FUNCTION_BLOCK FB_Machine_Run EXTENDS CycleHandleFB
VAR_INPUT
	Ctrl_ref:					REFERENCE TO Ctrl_Typ;
	 FB_RW_Ctrl_ref:			REFERENCE TO FB_RW_Ctrl;
END_VAR
VAR_OUTPUT
END_VAR
VAR
	MethInitDone:		BOOL;
	FB_HeaterProtection:FB_HeaterProtection;
END_VAR
VAR CONSTANT

// States are global
(*		
	MACHINE_RUN_INIT:						INT:=0;
	MACHINE_COLD_CUT_VALVE_OPEN:			INT:=10;
	MACHINE_WELD_VALVE_OPEN:				INT:=20;	
	MACHINE_HEATER_ON:						INT:=30;	
	MACHINE_HEATER_OFF:						INT:=40;
	MACHINE_VALVE_CLOSE:					INT:=50;	
	MACHINE_DONE:							INT:=100;	

*)

END_VAR

	IF NOT MethInitDone THEN
		MethInitDone	:= Meth_Init();
	END_IF
	
	
	IF  THIS^.CMD.Pause = FALSE THEN
		
		//-----------------------------
		//State Machine
		//-----------------------------
		CASE THIS^.StepNo OF
			MACHINE_RUN_INIT:
				IF THIS^.StepOneShotTrig THEN
					THIS^.Monitoring.StepMessage	:= 'Init: Start.';
					THIS^.Delay(IN:=FALSE);
					Meth_Rest_IO();
				ELSIF Meth_Enable(TRUE) THEN
					THIS^.StepNo	:= 	MACHINE_WAIT_DANCER_FULL;
				//	THIS^.StepNo	:= 	MACHINE_GRIPPER_END_POSITION;
				END_IF								
			
				
			MACHINE_WAIT_DANCER_FULL:
				IF THIS^.StepOneShotTrig THEN
					THIS^.Monitoring.StepMessage	:= 'Wait Dancer full';
					THIS^.Delay(IN:=FALSE);
				ELSIF Meth_WaitDancerFull(TRUE) THEN
					THIS^.StepNo	:= 	MACHINE_GRIPPER_RETRACT;
				END_IF					
								
	
			MACHINE_GRIPPER_RETRACT:
				IF THIS^.StepOneShotTrig THEN
					THIS^.Monitoring.StepMessage	:= 'Gripper retract';
					THIS^.Delay(IN:=FALSE);
					
				ELSIF Meth_gripperRetract(TRUE) THEN
					THIS^.StepNo	:= 	MACHINE_GRIPPER_END_POSITION;
				END_IF	

									
			MACHINE_GRIPPER_END_POSITION:
				IF THIS^.StepOneShotTrig THEN
					THIS^.Monitoring.StepMessage	:= 'Machine WAIT position';
					THIS^.Delay(IN:=FALSE);
				ELSIF Meth_gripperEndPosition(TRUE) THEN
					THIS^.StepNo	:= 	MACHINE_OUT_GRIPPER_START_POSITION;
				END_IF					
			
			MACHINE_OUT_GRIPPER_START_POSITION:
				IF THIS^.StepOneShotTrig THEN
					THIS^.Monitoring.StepMessage	:= 'Output Grippers to start position';
					Meth_OutGripperStartPos(FALSE) ;
				ELSIF Meth_OutGripperStartPos(TRUE) THEN
					THIS^.StepNo	:= 	MACHINE_OUT_GRIPPER_CLAMP;
				END_IF				
							
				
			MACHINE_OUT_GRIPPER_CLAMP:
				IF THIS^.StepOneShotTrig THEN
					THIS^.Monitoring.StepMessage	:= 'Machine grippers clamp';
					THIS^.Delay(IN:=FALSE);
				ELSIF Meth_OutGripperClamp(TRUE) THEN
					THIS^.StepNo	:= 	MACHINE_GRIPPER_OPEN;
				END_IF	
			

			MACHINE_GRIPPER_OPEN:
				IF THIS^.StepOneShotTrig THEN
					THIS^.Monitoring.StepMessage	:= 'Gripper Open';
					THIS^.Delay(IN:=FALSE);
				ELSIF Meth_gripperOpen(TRUE) THEN
					THIS^.StepNo	:= 	MACHINE_GRIPPER_START_POSITION;
				END_IF					
						
				
			MACHINE_GRIPPER_START_POSITION:
				IF THIS^.StepOneShotTrig THEN
					THIS^.Monitoring.StepMessage	:= 'Machine start position';
					THIS^.Delay(IN:=FALSE);
					
				ELSIF Meth_gripperStartPosition(TRUE) THEN
					THIS^.StepNo	:= 	MACHINE_GRIPPER_EXCTRACT;
				END_IF	
	
			
			MACHINE_GRIPPER_EXCTRACT:
			IF THIS^.StepOneShotTrig THEN
				THIS^.Monitoring.StepMessage	:= 'Gripper Extract';
				THIS^.Delay(IN:=FALSE);
			ELSIF Meth_gripperExtract(TRUE) THEN
				THIS^.StepNo	:= 	MACHINE_GRIPPER_CLOSE;
			END_IF				
				
			MACHINE_GRIPPER_CLOSE:
				IF THIS^.StepOneShotTrig THEN
					THIS^.Monitoring.StepMessage	:= 'Gripper Close';
					THIS^.Delay(IN:=FALSE);
				ELSIF Meth_gripperClose(TRUE) THEN
					THIS^.StepNo	:= 	MACHINE_COLD_CUT_VALVE_OPEN;
				END_IF	
	
			MACHINE_COLD_CUT_VALVE_OPEN:
				IF THIS^.StepOneShotTrig THEN
					THIS^.Monitoring.StepMessage	:= 'Cold cut valve open';
					THIS^.Delay(IN:=FALSE);
				ELSIF Meth_ColdCutValveOpen(TRUE) THEN
					THIS^.StepNo	:= 	MACHINE_WELD_VALVE_OPEN;
				END_IF	

			MACHINE_WELD_VALVE_OPEN://and gripper open
				IF THIS^.StepOneShotTrig THEN
					THIS^.Monitoring.StepMessage	:= 'Hot weld valve open press Down';
					THIS^.Delay(IN:=FALSE);
				ELSIF Meth_HotWeldValveOpen(TRUE) THEN
					THIS^.StepNo	:= 	MACHINE_HEATER_ON;
				END_IF					
				
			MACHINE_HEATER_ON://
				IF THIS^.StepOneShotTrig THEN
					THIS^.Monitoring.StepMessage	:= 'Heater ON';
					THIS^.Delay(IN:=FALSE);
				ELSIF Meth_HeaterON(TRUE) THEN
					THIS^.StepNo	:= 	MACHINE_HEATER_OFF;
				END_IF								
				
			MACHINE_HEATER_OFF://gripper retract
				IF THIS^.StepOneShotTrig THEN
					THIS^.Monitoring.StepMessage	:= 'Heater Off';
					THIS^.Delay(IN:=FALSE);
				ELSIF Meth_HeaterOff(TRUE) THEN
					THIS^.StepNo	:= 	MACHINE_CUT_WEB;
				END_IF					
						
			MACHINE_CUT_WEB:
				IF THIS^.StepOneShotTrig THEN
					THIS^.Monitoring.StepMessage	:= 'Close valves';
					THIS^.Delay(IN:=FALSE);
					gMachineCtrl.IO.Out.KniveCut:=NOT(gMachineCtrl.IO.Out.KniveCut);
				ELSIF Meth_CutWeb(TRUE) THEN
					THIS^.StepNo	:= 	MACHINE_VALVE_CLOSE;
				END_IF		
				
			MACHINE_VALVE_CLOSE:
				IF THIS^.StepOneShotTrig THEN
					THIS^.Monitoring.StepMessage	:= 'Close valves';
					THIS^.Delay(IN:=FALSE);
				ELSIF Meth_HeaterValvesClose(TRUE) THEN
					THIS^.StepNo	:= 	MACHINE_OUT_GRIPPER_END_POSITION;
				END_IF					
				
			MACHINE_OUT_GRIPPER_END_POSITION:
				IF THIS^.StepOneShotTrig THEN
					THIS^.Monitoring.StepMessage	:= 'Output Grippers to start position';
					Meth_OutGripperEndPos(FALSE) ;
				ELSIF Meth_OutGripperEndPos(TRUE) THEN
					THIS^.StepNo	:= 	MACHINE_DONE;
				END_IF								
				
			MACHINE_DONE:
				IF THIS^.StepOneShotTrig THEN
					THIS^.Monitoring.StepMessage	:= 'Machine cycle Done';
				ELSIF Meth_Done(TRUE) THEN
					THIS^.StepNo	:= 	MACHINE_RUN_INIT;
				END_IF			
			
				
			//UnUsed	
			
								
		END_CASE
	
	ELSE
		THIS^.Monitoring.StepMessage:= 'Pause';
		
		IF THIS^.Status.Fault = TRUE THEN
		//IF Meth_EmStop(TRUE) THEN
				THIS^.CMD.ResetCycle	:= TRUE;		// Reset the all state machine to start point
		//END_IF
			
		END_IF
		
	END_IF
	
	//============================================================================================
	// Reset Internal Function Blocks
	IF THIS^.CMD.ResetCycle = TRUE THEN
		IF FB_RW_Ctrl_ref.Running OR FB_RW_Ctrl_ref.Pause OR FB_RW_Ctrl_ref.Fault THEN
			FB_RW_Ctrl_ref.ResetCycle	:= TRUE;
		END_IF
	END_IF	
	
	THIS^.FB_HeaterProtection();
	THIS^.Delay();
	THIS^.CH_Logic();
	
	// Reset Meth_EmStop when at Init State
	IF THIS^.Pause = FALSE THEN
		//Meth_EmStop(FALSE);
	END_IF

METHOD PRIVATE Meth_ColdCutValveOpen : BOOL
VAR_INPUT
	Execute: 	BOOL;
END_VAR


	THIS^.Monitoring.StepMessage			:= 'Cold Cut Valve Open';
	THIS^.Monitoring.Error_Text				:= ' Fail';
	//THIS^.CMD.Deacivate_Sequence_Time_Out	:= TRUE;	// Disable time out to the all sequence
	THIS^.CMD.DeactivateStepTimeOut			:= TRUE;	// Disable time out to the actual step
	THIS^.Parameter.TimeOut					:= T#5S;


	
	gMachineCtrl.IO.Out.Buzzer	:=TRUE;
										
	THIS^.Delay.IN:=TRUE;
	THIS^.Delay.PT :=DINT_TO_TIME( Persist.PersistentStruct.TimeColdCutPressDown);// Ctrl_ref.Parameters.TimerPressDown1);
	IF THIS^.Delay.Q THEN
		Meth_ColdCutValveOpen	:= TRUE;
		gMachineCtrl.IO.Out.GripperOpen:=TRUE;
	END_IF
END_METHOD

METHOD Meth_CutWeb : BOOL
VAR_INPUT
	Execute: 	BOOL;
END_VAR
	THIS^.Monitoring.StepMessage			:= 'Cut Web';
	THIS^.Monitoring.Error_Text				:= ' Fail';
	//THIS^.CMD.Deacivate_Sequence_Time_Out	:= TRUE;	// Disable time out to the all sequence
	THIS^.CMD.DeactivateStepTimeOut			:= TRUE;	// Disable time out to the actual step
	THIS^.Parameter.TimeOut					:= T#5S;

	
											
	THIS^.Delay.IN:=TRUE;
	THIS^.Delay.PT :=DINT_TO_TIME( Persist.PersistentStruct.TimeKniveVut);// Ctrl_ref.Parameters.TimerPressDown1);
	IF THIS^.Delay.Q THEN
		Meth_CutWeb	:= TRUE;
		
		//gMachineCtrl.Parameters.UW_1_Param.EnableTension:=TRUE;
		//gMachineCtrl.Parameters.UW_2_Param.EnableTension:=TRUE;
		
	END_IF
END_METHOD

METHOD PRIVATE Meth_Done : BOOL
VAR_INPUT
	Execute: 	BOOL;
END_VAR


	//THIS^.Monitoring.StepMessage			:= 'Press 1 engage';
	//THIS^.Monitoring.Error_Text				:= 'Press 1 engage Fail';
	//THIS^.CMD.Deacivate_Sequence_Time_Out	:= TRUE;	// Disable time out to the all sequence
	//THIS^.CMD.DeactivateStepTimeOut			:= TRUE;	// Disable time out to the actual step
	//THIS^.Parameter.TimeOut					:= T#5S;

	//gMachineCtrl.Parameters.UW_1_Param.EnableDancer :=FALSE;
	//gMachineCtrl.Parameters.UW_2_Param.EnableDancer:=FALSE;	
	
	THIS^.Status.Done		:= TRUE;
	THIS^.Status.Running	:= FALSE;									
	Meth_Done	:= TRUE;
END_METHOD

METHOD PRIVATE Meth_Enable : BOOL
VAR_INPUT
	Execute: 	BOOL;
END_VAR


IF THIS^.CMD.Start THEN
	
	THIS^.Monitoring.StepMessage			:= 'Start';
	THIS^.Monitoring.Error_Text				:= 'Start Fail';
	THIS^.CMD.Deacivate_Sequence_Time_Out	:= TRUE;	// Disable time out to the all sequence
	THIS^.CMD.DeactivateStepTimeOut			:= TRUE;	// Disable time out to the actual step
	THIS^.Parameter.TimeOut					:= T#0.5S;

	THIS^.CMD.Start			:= FALSE;
	THIS^.Status.Done		:= FALSE;
	THIS^.Status.Running	:= TRUE;
	
	// Reset Commands and Statuses												
	
	Meth_Enable	:= TRUE;
END_IF
END_METHOD

METHOD PRIVATE Meth_gripperClose : BOOL
VAR_INPUT
	Execute: 	BOOL;
END_VAR


	THIS^.Monitoring.StepMessage			:= 'Gripper Close';
	THIS^.Monitoring.Error_Text				:= ' Fail';
	//THIS^.CMD.Deacivate_Sequence_Time_Out	:= TRUE;	// Disable time out to the all sequence
	THIS^.CMD.DeactivateStepTimeOut			:= TRUE;	// Disable time out to the actual step
	THIS^.Parameter.TimeOut					:= T#5S;

	gMachineCtrl.IO.Out.GripperOpen:=TRUE;
											
	THIS^.Delay.IN:=TRUE;
	THIS^.Delay.PT :=DINT_TO_TIME( Persist.PersistentStruct.TimeGripperOpen);// Ctrl_ref.Parameters.TimerPressDown1);
	IF THIS^.Delay.Q THEN
		Meth_gripperClose	:= TRUE;
		
		//gMachineCtrl.Parameters.UW_1_Param.EnableTension:=TRUE;
		//gMachineCtrl.Parameters.UW_2_Param.EnableTension:=TRUE;
		
	END_IF
END_METHOD

METHOD PRIVATE Meth_gripperEndPosition : BOOL
VAR_INPUT
	Execute: 	BOOL;
END_VAR


	//THIS^.Monitoring.StepMessage			:= 'GripperStartPosition';
	THIS^.Monitoring.Error_Text				:= ' Fail';
	//THIS^.CMD.Deacivate_Sequence_Time_Out	:= TRUE;	// Disable time out to the all sequence
	THIS^.CMD.DeactivateStepTimeOut			:= TRUE;	// Disable time out to the actual step
	THIS^.Parameter.TimeOut					:= T#5S;

	gMachineCtrl.IO.Out.GripperPistonPosition:=TRUE;
	
	gMachineCtrl.IO.Out.ExternalNipMotor:=TRUE;
		
	//gMachineCtrl.Parameters.UW_1_Param.kp := gMachineCtrl.Parameters.UW_1_Param.kpMove;
	////gMachineCtrl.Parameters.UW_1_Param.TN := gMachineCtrl.Parameters.UW_1_Param.TNMove;
	//.Parameters.UW_2_Param.kp := gMachineCtrl.Parameters.UW_2_Param.kpMove;
	//gMachineCtrl.Parameters.UW_2_Param.TN := gMachineCtrl.Parameters.UW_2_Param.TNMove;



							
	THIS^.Delay.IN:=TRUE;
	THIS^.Delay.PT :=DINT_TO_TIME( Persist.PersistentStruct.TimeGripperStartPosition);// Ctrl_ref.Parameters.TimerPressDown1);
	IF THIS^.Delay.Q THEN
		Meth_gripperEndPosition	:= TRUE;
		
	//.Parameters.UW_1_Param.kp := 0.1;
	//gMachineCtrl.Parameters.UW_1_Param.TN := T#0MS;
	//gMachineCtrl.Parameters.UW_2_Param.kp := 0.1;
	//gMachineCtrl.Parameters.UW_2_Param.TN := T#0MS;			
	
	gMachineCtrl.IO.Out.ExternalNipMotor:=FALSE;
		
	END_IF
END_METHOD

METHOD PRIVATE Meth_gripperExtract : BOOL
VAR_INPUT
	Execute: 	BOOL;
END_VAR


	//THIS^.Monitoring.StepMessage			:= 'Gripper Retract';
	THIS^.Monitoring.Error_Text				:= ' Fail';
	//THIS^.CMD.Deacivate_Sequence_Time_Out	:= TRUE;	// Disable time out to the all sequence
	THIS^.CMD.DeactivateStepTimeOut			:= TRUE;	// Disable time out to the actual step
	THIS^.Parameter.TimeOut					:= T#5S;

	gMachineCtrl.IO.Out.GripperRetract:=TRUE;
											
	THIS^.Delay.IN:=TRUE;
	THIS^.Delay.PT :=DINT_TO_TIME( Persist.PersistentStruct.TimeGripperRetract);// Ctrl_ref.Parameters.TimerPressDown1);
	IF THIS^.Delay.Q THEN
		Meth_gripperExtract	:= TRUE;
	END_IF
END_METHOD

METHOD PRIVATE Meth_gripperOpen : BOOL
VAR_INPUT
	Execute: 	BOOL;
END_VAR


	//THIS^.Monitoring.StepMessage			:= 'Gripper Open';
	THIS^.Monitoring.Error_Text				:= ' Fail';
	//THIS^.CMD.Deacivate_Sequence_Time_Out	:= TRUE;	// Disable time out to the all sequence
	THIS^.CMD.DeactivateStepTimeOut			:= TRUE;	// Disable time out to the actual step
	THIS^.Parameter.TimeOut					:= T#5S;

	gMachineCtrl.IO.Out.GripperOpen:=FALSE;
											
	THIS^.Delay.IN:=TRUE;
	THIS^.Delay.PT :=DINT_TO_TIME( Persist.PersistentStruct.TimeGripperOpen);// Ctrl_ref.Parameters.TimerPressDown1);
	IF THIS^.Delay.Q THEN
		Meth_gripperOpen	:= TRUE;
	END_IF
END_METHOD

METHOD PRIVATE Meth_gripperRetract : BOOL
VAR_INPUT
	Execute: 	BOOL;
END_VAR


	//THIS^.Monitoring.StepMessage			:= 'Gripper Retract';
	THIS^.Monitoring.Error_Text				:= ' Fail';
	//THIS^.CMD.Deacivate_Sequence_Time_Out	:= TRUE;	// Disable time out to the all sequence
	THIS^.CMD.DeactivateStepTimeOut			:= TRUE;	// Disable time out to the actual step
	THIS^.Parameter.TimeOut					:= T#5S;

	gMachineCtrl.IO.Out.GripperRetract:=FALSE;
											
	THIS^.Delay.IN:=TRUE;
	THIS^.Delay.PT :=DINT_TO_TIME( Persist.PersistentStruct.TimeGripperRetract);// Ctrl_ref.Parameters.TimerPressDown1);
	IF THIS^.Delay.Q THEN
		Meth_gripperRetract	:= TRUE;
	END_IF
END_METHOD

METHOD PRIVATE Meth_gripperStartPosition : BOOL
VAR_INPUT
	Execute: 	BOOL;
END_VAR


	//THIS^.Monitoring.StepMessage			:= 'GripperStartPosition';
	THIS^.Monitoring.Error_Text				:= ' Fail';
	//THIS^.CMD.Deacivate_Sequence_Time_Out	:= TRUE;	// Disable time out to the all sequence
	THIS^.CMD.DeactivateStepTimeOut			:= TRUE;	// Disable time out to the actual step
	THIS^.Parameter.TimeOut					:= T#5S;

	gMachineCtrl.IO.Out.GripperPistonPosition:=FALSE;
											
	THIS^.Delay.IN:=TRUE;
	THIS^.Delay.PT :=DINT_TO_TIME( Persist.PersistentStruct.TimeGripperHomePosition);// Ctrl_ref.Parameters.TimerPressDown1);
	IF THIS^.Delay.Q THEN
		Meth_gripperStartPosition	:= TRUE;
	END_IF
END_METHOD

METHOD PRIVATE Meth_HeaterOff : BOOL
VAR_INPUT
	Execute: 	BOOL;
END_VAR


	THIS^.Monitoring.StepMessage			:= 'Heater Off';
	THIS^.Monitoring.Error_Text				:= ' Heater Off Fail';
	//THIS^.CMD.Deacivate_Sequence_Time_Out	:= TRUE;	// Disable time out to the all sequence
	THIS^.CMD.DeactivateStepTimeOut			:= TRUE;	// Disable time out to the actual step
	THIS^.Parameter.TimeOut					:= T#5S;

	
											
	THIS^.Delay.IN:=TRUE;
	THIS^.Delay.PT :=DINT_TO_TIME( Persist.PersistentStruct.TimerHotWeldingOff);// Ctrl_ref.Parameters.TimerPressDown1);
	IF THIS^.Delay.Q AND THIS^.FB_HeaterProtection.Done THEN
		Meth_HeaterOff	:= TRUE;
	END_IF
END_METHOD

METHOD PRIVATE Meth_HeaterON : BOOL
VAR_INPUT
	Execute: 	BOOL;
END_VAR


	THIS^.Monitoring.StepMessage			:= 'Heater ON';
	THIS^.Monitoring.Error_Text				:= ' Heater ON Fail';
	//THIS^.CMD.Deacivate_Sequence_Time_Out	:= TRUE;	// Disable time out to the all sequence
	THIS^.CMD.DeactivateStepTimeOut			:= TRUE;	// Disable time out to the actual step
	THIS^.Parameter.TimeOut					:= T#5S;

	//Ctrl_ref.IO.Out.HeaterOn := TRUE;
	FB_HeaterProtection.Excute:=TRUE;
			
	gMachineCtrl.IO.Out.ColdCutPistonDown:=TRUE;						
//	THIS^.Delay.IN:=TRUE;
//	THIS^.Delay.PT :=DINT_TO_TIME( Persist.PersistentStruct.TimerHotWeldingOn);// Ctrl_ref.Parameters.TimerPressDown1);
//	IF THIS^.Delay.Q THEN
		Meth_HeaterON	:= TRUE;;
//	END_IF
END_METHOD

METHOD PRIVATE Meth_HeaterValvesClose : BOOL
VAR_INPUT
	Execute: 	BOOL;
END_VAR


	THIS^.Monitoring.StepMessage			:= 'Valves close';
	THIS^.Monitoring.Error_Text				:= ' Valves close Fail';
	//THIS^.CMD.Deacivate_Sequence_Time_Out	:= TRUE;	// Disable time out to the all sequence
	THIS^.CMD.DeactivateStepTimeOut			:= TRUE;	// Disable time out to the actual step
	THIS^.Parameter.TimeOut					:= T#5S;

	gMachineCtrl.IO.Out.PressDown:=FALSE;
	gMachineCtrl.IO.Out.ColdCutPistonDown:=FALSE;										
	THIS^.Delay.IN:=TRUE;
	THIS^.Delay.PT :=DINT_TO_TIME( Persist.PersistentStruct.TimerPressUp);// Ctrl_ref.Parameters.TimerPressDown1);
	IF THIS^.Delay.Q THEN
		Meth_HeaterValvesClose	:= TRUE;
	END_IF
END_METHOD

METHOD PRIVATE Meth_HotWeldValveOpen : BOOL
VAR_INPUT
	Execute: 	BOOL;
END_VAR


	THIS^.Monitoring.StepMessage			:= 'Hot Weld Valve Open';
	THIS^.Monitoring.Error_Text				:= ' Hot Weld Valve Open Fail';
	//THIS^.CMD.Deacivate_Sequence_Time_Out	:= TRUE;	// Disable time out to the all sequence
	THIS^.CMD.DeactivateStepTimeOut			:= TRUE;	// Disable time out to the actual step
	THIS^.Parameter.TimeOut					:= T#5S;

	gMachineCtrl.IO.Out.PressDown :=TRUE;
											
	THIS^.Delay.IN:=TRUE;
	THIS^.Delay.PT :=DINT_TO_TIME( Persist.PersistentStruct.TimeHotWeldPressDown);// Ctrl_ref.Parameters.TimerPressDown1);
	IF THIS^.Delay.Q THEN
		Meth_HotWeldValveOpen	:= TRUE;
		gMachineCtrl.IO.Out.Buzzer	:=FALSE;
	END_IF
END_METHOD

METHOD Meth_Init :BOOL
VAR_INPUT
END_VAR
Meth_Init:=TRUE;
END_METHOD

METHOD PRIVATE Meth_MororON : BOOL
VAR_INPUT
	Execute: 	BOOL;
END_VAR


	THIS^.Monitoring.StepMessage			:= 'Motor ON';
	THIS^.Monitoring.Error_Text				:= ' Motor ON Fail';
	//THIS^.CMD.Deacivate_Sequence_Time_Out	:= TRUE;	// Disable time out to the all sequence
	THIS^.CMD.DeactivateStepTimeOut			:= TRUE;	// Disable time out to the actual step
	THIS^.Parameter.TimeOut					:= T#5S;


											
	THIS^.Delay.IN:=TRUE;
	THIS^.Delay.PT :=DINT_TO_TIME( Persist.PersistentStruct.TimerMotorOn);// Ctrl_ref.Parameters.TimerPressDown1);
	IF THIS^.Delay.Q  AND FB_RW_Ctrl_ref.Done THEN
		Meth_MororON	:= TRUE;
	END_IF
END_METHOD

METHOD Meth_OutGripperClamp : BOOL
VAR_INPUT
	Execute: 	BOOL;
END_VAR


	THIS^.Monitoring.StepMessage			:= 'Output Gripper Close';
	THIS^.Monitoring.Error_Text				:= ' Fail';
	//THIS^.CMD.Deacivate_Sequence_Time_Out	:= TRUE;	// Disable time out to the all sequence
	THIS^.CMD.DeactivateStepTimeOut			:= TRUE;	// Disable time out to the actual step
	THIS^.Parameter.TimeOut					:= T#5S;

	gMachineCtrl.IO.Out.Output_GripperClose:=TRUE;
											
	THIS^.Delay.IN:=TRUE;
	THIS^.Delay.PT :=DINT_TO_TIME( Persist.PersistentStruct.TimeOutputGripperClose);// Ctrl_ref.Parameters.TimerPressDown1);
	IF THIS^.Delay.Q THEN
		Meth_OutGripperClamp	:= TRUE;
		
		//gMachineCtrl.Parameters.UW_1_Param.EnableTension:=TRUE;
		//gMachineCtrl.Parameters.UW_2_Param.EnableTension:=TRUE;
		
	END_IF
END_METHOD

METHOD Meth_OutGripperEndPos : BOOL
VAR_INPUT
	Execute: 	BOOL;
END_VAR
VAR_INST
	ExecuteTrig: 	Trigger;
END_VAR




IF ExecuteTrig.EDGEPOS(Execute) THEN
	Meth_OutGripperEndPos:=	FALSE;
	THIS^.SubStepNo:= 	1;	
END_IF

IF ExecuteTrig.EDGENEG(Execute) THEN
	Meth_OutGripperEndPos:=	FALSE;
END_IF

CASE THIS^.SubStepNo OF
	(* Power ON*)
	1:
		THIS^.Monitoring.StepMessage	:= 'Move output gripper to end';								
		gWebAxes.Output.Crtl.Basic_axis.Input.Command.MoveAbsolute		:= TRUE;
		gWebAxes.Output.Crtl.Basic_axis.Input.Parameter.Velocity		:= 500;//mm/sec
		gWebAxes.Output.Crtl.Basic_axis.Input.Parameter.Position		:= gMachineCtrl.Parameters.OutgripperEndPosition;//mm
		
		THIS^.SubStepNo:= 2;		
	
	2:	
		THIS^.Monitoring.StepMessage:= 'Wait output gripper end';
		
		IF gWebAxes.Output.Crtl.Basic_axis.Output.monitor.ActPosition > (gMachineCtrl.Parameters.OutgripperEndPosition-200) THEN
			gMachineCtrl.IO.Out.Output_GripperClose:=FALSE;
		END_IF
							
		IF gWebAxes.Output.Crtl.Basic_axis.Output.Status.MC_MoveAbsolut.Done THEN
			THIS^.SubStepNo	:= 3 ;
		END_IF
		
	3:	
		THIS^.Monitoring.StepMessage	:= 'Move output gripper to end';								
		gWebAxes.Output.Crtl.Basic_axis.Input.Command.MoveAbsolute		:= TRUE;
		gWebAxes.Output.Crtl.Basic_axis.Input.Parameter.Velocity		:= 100;//mm/sec
		gWebAxes.Output.Crtl.Basic_axis.Input.Parameter.Position		:= gMachineCtrl.Parameters.OutgripperEndPosition+200;//mm
		
		THIS^.SubStepNo:= 4;	
				
	4:	
		THIS^.Monitoring.StepMessage:= 'Wait output gripper end';
							
		IF gWebAxes.Output.Crtl.Basic_axis.Output.Status.MC_MoveAbsolut.Done THEN
			THIS^.SubStepNo	:= 100 ;
			Meth_OutGripperEndPos:=	TRUE;
		END_IF							
END_CASE
END_METHOD

METHOD Meth_OutGripperStartPos : BOOL
VAR_INPUT
	Execute: 	BOOL;
END_VAR
VAR_INST
	ExecuteTrig: 	Trigger;
END_VAR




IF ExecuteTrig.EDGEPOS(Execute) THEN
	Meth_OutGripperStartPos:=	FALSE;
	THIS^.SubStepNo:= 	1;	
END_IF

IF ExecuteTrig.EDGENEG(Execute) THEN
	Meth_OutGripperStartPos:=	FALSE;
END_IF

CASE THIS^.SubStepNo OF
	(* Power ON*)
	1:
		THIS^.Monitoring.StepMessage	:= 'Move output gripper to home';								
		gWebAxes.Output.Crtl.Basic_axis.Input.Command.MoveAbsolute		:= TRUE;
		gWebAxes.Output.Crtl.Basic_axis.Input.Parameter.Velocity		:= 500;//mm/sec
		gWebAxes.Output.Crtl.Basic_axis.Input.Parameter.Position		:= 0;
		
		THIS^.SubStepNo:= 2;		
	
	2:	
		THIS^.Monitoring.StepMessage:= 'Wait output gripper home';
									
		IF gWebAxes.Output.Crtl.Basic_axis.Output.Status.MC_MoveAbsolut.Done THEN
			THIS^.SubStepNo	:= 3 ;
			Meth_OutGripperStartPos	:= TRUE;
		END_IF
		

							
END_CASE
END_METHOD

METHOD Meth_Rest_IO 
VAR_INPUT
	
END_VAR

Ctrl_ref.IO.Out.HeaterOn := FALSE;
END_METHOD

METHOD PRIVATE Meth_WaitDancerFull : BOOL
VAR_INPUT
	Execute: 	BOOL;
END_VAR


	//THIS^.Monitoring.StepMessage			:= 'Gripper Retract';
	THIS^.Monitoring.Error_Text				:= ' Fail';
	//THIS^.CMD.Deacivate_Sequence_Time_Out	:= TRUE;	// Disable time out to the all sequence
	THIS^.CMD.DeactivateStepTimeOut			:= TRUE;	// Disable time out to the actual step
	THIS^.Parameter.TimeOut					:= T#5S;

	gMachineCtrl.Parameters.UW_1_Param.EnableDancer :=TRUE;
	gMachineCtrl.Parameters.UW_2_Param.EnableDancer:=TRUE;
											
	THIS^.Delay.IN:=TRUE;
	THIS^.Delay.PT :=DINT_TO_TIME( Persist.PersistentStruct.TimeGripperRetract);// Ctrl_ref.Parameters.TimerPressDown1);
	IF  (gMachineCtrl.Status.UW_1_DancerFull 
	AND gMachineCtrl.Status.UW_2_DancerFull)
	OR gMachineCtrl.Simulation THEN
		Meth_WaitDancerFull	:= TRUE;
	END_IF
END_METHOD

END_FUNCTION_BLOCK

(* stored: Version 1.1.0.1, ProductVersion 3.1.4024.3
   POU FB_Machine_Run: Id {a35008fa-9a47-43bf-8bba-12b194395176}, SpecialFunc None
   Folder Output: Id {dac0a439-9dfa-42c6-a811-39bb8546ae29}
   Method Meth_ColdCutValveOpen: Id {38048cc7-a9cb-4ee7-b874-5ec149a94069}
   Method Meth_CutWeb: Id {211628b9-63a3-4bcc-ac4e-3e809fb7de14}
   Method Meth_Done: Id {dc153501-6cca-42a0-82d9-0d52ed4c6e43}
   Method Meth_Enable: Id {b5be41ac-744e-4679-94f1-8dfb217df25b}
   Method Meth_gripperClose: Id {37507847-a2b3-49e7-ba5f-b366e3c22d51}
   Method Meth_gripperEndPosition: Id {a8b7c3d8-74eb-4445-8e48-dcabaa2a591a}
   Method Meth_gripperExtract: Id {88b82776-2d79-439b-b194-70d1d3083bef}
   Method Meth_gripperOpen: Id {f6a1064a-5131-430d-8367-ccb407406c03}
   Method Meth_gripperRetract: Id {d06a811c-5b63-42cb-b4a6-dd444d5db989}
   Method Meth_gripperStartPosition: Id {5480c9df-d06a-4df1-b021-6968e1c8639e}
   Method Meth_HeaterOff: Id {8e306fcf-d1b3-486d-b339-3b5cb7d038c0}
   Method Meth_HeaterON: Id {7ec11b00-92d9-4b61-981f-289b0ad43042}
   Method Meth_HeaterValvesClose: Id {82a40b60-a497-49ed-a5e1-19b1d9212e56}
   Method Meth_HotWeldValveOpen: Id {ba5ea5f4-56c3-4cce-87ed-53b8215badee}
   Method Meth_Init: Id {5c76d4f9-85c8-4033-af06-e822798f3ddf}
   Method Meth_MororON: Id {16058515-1409-40f5-860f-8187b9ce333e}
   Method Meth_OutGripperClamp: Id {711cba81-d1b0-4884-8164-cc610faa3464}
   Method Meth_OutGripperEndPos: Id {2c9b30d7-a32c-4725-b860-4530713ad592}
   Method Meth_OutGripperStartPos: Id {d72cd012-3474-48ca-8377-114a9a5f491b}
   Method Meth_Rest_IO: Id {959d1cc9-2dae-4247-ae06-4d56dd20472c}
   Method Meth_WaitDancerFull: Id {3881fe4d-5207-496a-98cf-763cf23fb35a} *)
